TYPE ST_TuneParams :
STRUCT
	fKp			:LREAL;
	fTn			:LREAL;
	fTv			:LREAL;
	fTd			:LREAL;
END_STRUCT
END_TYPE

(* stored: Version 1.1.0.1, ProductVersion 3.1.4024.11
   DUT ST_TuneParams: Id {10007334-1ba9-0cf5-262c-ee0524cac7cb} *)
